// TIA Portal V17 export
// export: Created 2023-12-22T15:08:09.4303305Z, ExportSetting WithDefaults, DisplayName Totally Integrated Automation Portal, DisplayVersion V17, DisplayName TIA Portal Openness, DisplayVersion V17, DisplayName TIA Portal Version Control Interface, DisplayVersion V17, DisplayName STEP 7 Professional, DisplayVersion V17, DisplayName STEP 7 Safety, DisplayVersion V17, DisplayName WinCC Advanced, DisplayVersion V17
DATA_BLOCK "ModBus_RTU_DB"   // DB30
VERSION : 0.1
// stored: AutoNumber false, DBAccessibleFromOPCUA true, DBAccessibleFromWebserver true, InstanceOfName ModBus_RTU, InstanceOfType FB
"ModBus_RTU"
   // VAR RETAIN
   //    DATA : Array[0..100] of Word;
   //    "Step" : Int;
   //    Device : Int;
   //    Limit { S7_SetPoint := 'True'} : Int := 10;
   //    COM_Config : Struct
   //       Baud_Rate { S7_SetPoint := 'True'} : UDInt := 115200;
   //       Port { S7_SetPoint := 'True'} : PORT := 0;
   //    END_STRUCT;
   //    COM_Control : Struct
   //       Enable { S7_SetPoint := 'True'} : Bool := TRUE;
   //       Start : Bool;
   //       Reset : Bool;
   //       Load_Done : Bool;
   //       Load_Status : Word;
   //       REQ_Done : Bool;
   //       REQ_Busy : Bool;
   //       REQ_Error : Bool;
   //       REQ_Status : Word;
   //       Error_Code : Word;
   //       Status : Int;
   //    END_STRUCT;
   //    COM_REQ : Struct
   //       ADDR : UInt;
   //       MODE : USInt;
   //       Register : UDInt;
   //       Length : UInt;
   //    END_STRUCT;
   //    DEV_Config : Array[1..10] of Struct
   //       Use { S7_SetPoint := 'True'} : Bool;
   //       MODE { S7_SetPoint := 'True'} : Bool;
   //       ADDR { S7_SetPoint := 'True'} : UInt;
   //       Register { S7_SetPoint := 'True'} : UDInt;
   //       Length { S7_SetPoint := 'True'} : UInt;
   //       Source_DB { S7_SetPoint := 'True'} : UInt;
   //       Source_OFFSET { S7_SetPoint := 'True'} : UInt;
   //       Target_DB { S7_SetPoint := 'True'} : UInt;
   //       Target_OFFSET { S7_SetPoint := 'True'} : UInt;
   //       Status : UInt;
   //    END_STRUCT;
   //    MB_COMM_LOAD { S7_SetPoint := 'True'} : Modbus_Comm_Load;
   //    MB_MASTER { S7_SetPoint := 'True'} : Modbus_Master;
   //    T_Busy : "Time_M";
   // END_VAR
BEGIN
   DEV_Config[1..10].Use := FALSE;
   DEV_Config[1..10].MODE := FALSE;
   DEV_Config[1..10].ADDR := 0;
   DEV_Config[1..10].Register := 0;
   DEV_Config[1..10].Length := 0;
   DEV_Config[1..10].Source_DB := 0;
   DEV_Config[1..10].Source_OFFSET := 0;
   DEV_Config[1..10].Target_DB := 0;
   DEV_Config[1..10].Target_OFFSET := 0;
END_DATA_BLOCK
